PROGRAM Stn055_56_StorageBypassMainMergePrestopBlu
VAR
	{attribute 'TcLinkToOSO' := '.iPuckPresent   :=  <0,1,3>TIIB[N12S00 (AL1332)]^N12S05 (AL2341)^TxPDO^input byte 0;
								 .iBufferFull  :=  <0,1,3>TIIB[N12S00 (AL1332)]^N12S05 (AL2341)^TxPDO^input byte 2;
								 .oStopLower   :=  <0,1,4>TIIB[N12S00 (AL1332)]^N12S02 (EX260)^RxPDO^output byte 2'}
	fbConvStop: FB_ConvStop;
	
END_VAR

//  This code instantiates a component that is implimented as a common function block
//    Note that I/O is linked directly to I/O variables inside the named instance

gStn055_56_StorageBypassMainMergePrestopBlu.ConvRunning := gConsumed_SafetyInterfaceConv.MtrRunning.Enc051Mtr03;

fbConvStop(
	pStn := ADR(gStn055),
	pCmp := ADR(gStn055_56_StorageBypassMainMergePrestopBlu),
	pUpstreamStop := 0,
	pStateTraceBuffer := ADR(gStn055_StateTraceBuffer),
	pStateTraceFifo := ADR(gStn055_StateTraceFifo),
	pStats := ADR(gStn055_02_Stats));

END_PROGRAM

(* stored: Version 1.1.0.1, ProductVersion 3.1.4024.6
   POU Stn055_56_StorageBypassMainMergePrestopBlu: Id {40cfbcb6-62a1-4ccc-b193-995e0d7bf464}, SpecialFunc None *)
